// TIA Portal V17 export
// export: Created 2021-12-29T14:14:50.3702334Z, ExportSetting WithDefaults, DisplayName Totally Integrated Automation Portal, DisplayVersion V17, DisplayName TIA Portal Openness, DisplayVersion V17, DisplayName TIA Portal Version Control Interface, DisplayVersion V17, DisplayName STEP 7 Professional, DisplayVersion V17, DisplayName STEP 7 Safety, DisplayVersion V17, DisplayName WinCC Professional, DisplayVersion V17
DATA_BLOCK "DB_Tolvas"   // DB5
VERSION : 0.1
// stored: AutoNumber true, DBAccessibleFromOPCUA true, DBAccessibleFromWebserver true, InstanceOfName FB_Tolvas, InstanceOfType FB
"FB_Tolvas"
   // VAR
   //    "Timer" : "Clase_Tolvas";
   // END_VAR
BEGIN
END_DATA_BLOCK
